// TwinCAT 3 PLC project Portal
// ProgramVersion: 3.1.4024.0
// libraries:
//   Tc2_Drive, * (Beckhoff Automation GmbH)
//   Tc2_EtherCAT, * (Beckhoff Automation GmbH)
//   Tc2_Standard, * (Beckhoff Automation GmbH)
//   Tc2_System, * (Beckhoff Automation GmbH)
//   Tc2_Utilities, * (Beckhoff Automation GmbH)
//   Tc3_Module, * (Beckhoff Automation GmbH)
// project tree:
//   DUTs/ PanelButton.TcDUT, StateMachine.TcDUT
//   POUs/ RPC_PanelProcess.TcPOU, RPC_ScopeProcess.TcPOU, RPC_SoEProcess.TcPOU, MAIN.TcPOU
//   Scope/ FB_ExportScopeData.TcPOU, FB_GenerateFileSuffixByTime.TcPOU, FB_ScopeServer.TcPOU
//   GVLs/ GlobalVar.TcGVL
//   / PlcTask.TcTTO
// real-time tasks:
//   TASK PlcTask: cycle T#250us, priority 10, ADS port 350
//   TASK MotionControl: cycle T#250us, priority 4, ADS port 352
//   TASK ModuleSpindle: cycle T#250us, priority 6, ADS port 351
//   TASK ModuleAxisGroup: cycle T#250us, priority 8, ADS port 353
//   TASK ModuleTest: cycle T#250us, priority 12, ADS port 354
//   TASK TestHMI: cycle T#10ms, priority 18, ADS port 355
//   TASK ModuleSafety: cycle T#250us, priority 14, ADS port 356
// I/O:
//   DEVICE BeckhoffBench, AmsNetId 169.254.41.58.4.1
//     ZY [AX5201-0000-0214 EtherCAT Drive (SoE, 2 Ch.)]
//     Gantry [AX5201-0000-0214 EtherCAT Drive (SoE, 2 Ch.)]
//     Panel [iA-MPA64B0 2xMII_REV00030022]
//     Drive 4 (MCDLN35BE) [MCDLN35BE]
// variable links:
//   Portal/Portal Instance <-> BeckhoffBench/Gantry
//     PlcTask Inputs/MAIN.rpc_SoEProcess.stPlcDriveRef[0]/aNetId <-> InfoData/AdsAddr/netId
//     PlcTask Inputs/MAIN.rpc_SoEProcess.stPlcDriveRef[1]/aNetId <-> InfoData/AdsAddr/netId
//     PlcTask Inputs/MAIN.rpc_SoEProcess.stPlcDriveRef[0]/nDriveNo <-> InfoData/Chn1
//     PlcTask Inputs/MAIN.rpc_SoEProcess.stPlcDriveRef[1]/nDriveNo <-> InfoData/Chn0
//     PlcTask Inputs/MAIN.rpc_SoEProcess.stPlcDriveRef[0]/nSlaveAddr <-> InfoData/AdsAddr/port
//     PlcTask Inputs/MAIN.rpc_SoEProcess.stPlcDriveRef[1]/nSlaveAddr <-> InfoData/AdsAddr/port
//   Portal/Portal Instance <-> BeckhoffBench/Panel
//     PlcTask Inputs/MAIN.rpc_PanelProcess.handwheelCurrPos <-> PANEL_Inputs/TEACH_HANDWHEEL
//     PlcTask Inputs/MAIN.rpc_PanelProcess.pInput[0] <-> PANEL_Inputs/PIO_IN1
//     PlcTask Inputs/MAIN.rpc_PanelProcess.pInput[1] <-> PANEL_Inputs/PIO_IN2
//     PlcTask Inputs/MAIN.rpc_PanelProcess.pInput[2] <-> PANEL_Inputs/PIO_IN3
//     PlcTask Inputs/MAIN.rpc_PanelProcess.pInput[3] <-> PANEL_Inputs/PIO_IN4
//     PlcTask Inputs/MAIN.rpc_PanelProcess.pInput[4] <-> PANEL_Inputs/PIO_IN5
//     PlcTask Inputs/MAIN.rpc_PanelProcess.pInput[5] <-> PANEL_Inputs/PIO_IN7
//     PlcTask Outputs/MAIN.rpc_PanelProcess.pOutput[0] <-> PANEL_Outputs/PIO_OUT1
//     PlcTask Outputs/MAIN.rpc_PanelProcess.pOutput[1] <-> PANEL_Outputs/PIO_OUT2
//     PlcTask Outputs/MAIN.rpc_PanelProcess.pOutput[2] <-> PANEL_Outputs/PIO_OUT3
//     PlcTask Outputs/MAIN.rpc_PanelProcess.pOutput[3] <-> PANEL_Outputs/PIO_OUT4
//     PlcTask Outputs/MAIN.rpc_PanelProcess.pOutput[4] <-> PANEL_Outputs/PIO_OUT5
//     PlcTask Outputs/MAIN.rpc_PanelProcess.pOutput[5] <-> PANEL_Outputs/PIO_OUT7
//   Portal/Portal Instance <-> BeckhoffBench/ZY
//     PlcTask Inputs/MAIN.rpc_SoEProcess.stPlcDriveRef[2]/aNetId <-> InfoData/AdsAddr/netId
//     PlcTask Inputs/MAIN.rpc_SoEProcess.stPlcDriveRef[3]/aNetId <-> InfoData/AdsAddr/netId
//     PlcTask Inputs/MAIN.rpc_SoEProcess.stPlcDriveRef[2]/nDriveNo <-> InfoData/Chn1
//     PlcTask Inputs/MAIN.rpc_SoEProcess.stPlcDriveRef[3]/nDriveNo <-> InfoData/Chn0
//     PlcTask Inputs/MAIN.rpc_SoEProcess.stPlcDriveRef[2]/nSlaveAddr <-> InfoData/AdsAddr/port
//     PlcTask Inputs/MAIN.rpc_SoEProcess.stPlcDriveRef[3]/nSlaveAddr <-> InfoData/AdsAddr/port
//   Portal/Portal Instance <-> MotionControl/MotionControl_Obj1 (MotionControl)
//     PlcTask Outputs/MAIN.rpc_PanelProcess.objID <-> Inputs/OidPanelProcess
//     PlcTask Outputs/MAIN.rpc_PanelProcess.panelInfoOutput <-> Inputs/PanelInformation
//     PlcTask Outputs/MAIN.rpc_ScopeProcess.objID <-> Inputs/OidScopeProcess
//   Portal/Portal Instance <-> MotionControl/MotionControl_Obj3 (ModuleAxisGroup)
//     PlcTask Outputs/MAIN.rpc_SoEProcess.objID <-> Inputs/OidSoEProcess
//   MotionControl/MotionControl_Obj1 (MotionControl) <-> MotionControl/MotionControl_Obj3 (ModuleAxisGroup)
//     Outputs/ContinuousMovingCommand <-> Inputs/ContinuousMovingCommand
//     Outputs/ManualMovingCommand <-> Inputs/ManualMovingCommand
//   MotionControl/MotionControl_Obj1 (MotionControl) <-> MotionControl/MotionControl_Obj4 (ModuleSafety)
//     Inputs/ErrorCode <-> Outputs/ErrorCode
//   MotionControl/MotionControl_Obj2 (ModuleSpindle) <-> MotionControl/MotionControl_Obj4 (ModuleSafety)
//     Outputs/SpindleInfo <-> Inputs/DiagnosticInfo/SpindleInfo
//     Outputs/StateSpindle <-> Inputs/DiagnosticInfo/StateSpindle
//   MotionControl/MotionControl_Obj3 (ModuleAxisGroup) <-> MotionControl/MotionControl_Obj4 (ModuleSafety)
//     Outputs/AxisGroupInfo <-> Inputs/DiagnosticInfo/AxisGroupInfo
//     Outputs/StateAxisGroup <-> Inputs/DiagnosticInfo/StateAxisGroup
//   (this object) <-> MotionControl/MotionControl_Obj2 (ModuleSpindle)
//     Drive 4 (MCDLN35BE)/Receive PDO mapping 1/Controlword <-> Outputs/SpindleOutput/ControlWord
//     Drive 4 (MCDLN35BE)/Receive PDO mapping 1/Modes of operation <-> Outputs/SpindleOutput/OperationMode
//     Drive 4 (MCDLN35BE)/Receive PDO mapping 1/Target position <-> Outputs/SpindleOutput/TargetPosition
//     Drive 4 (MCDLN35BE)/Transmit PDO mapping 1/Modes of operation display <-> Inputs/SpindleInput/ActualOpMode
//     Drive 4 (MCDLN35BE)/Transmit PDO mapping 1/Position actual value <-> Inputs/SpindleInput/ActualAbsPos
//     Drive 4 (MCDLN35BE)/Transmit PDO mapping 1/Statusword <-> Inputs/SpindleInput/StatusWord
//   (this object) <-> MotionControl/MotionControl_Obj3 (ModuleAxisGroup)
//     Gantry/AT 1/Class 1 diagnostic (C1D) <-> Inputs/AxisInputs[1]/ErrorCode
//     Gantry/AT 2/Class 1 diagnostic (C1D) <-> Inputs/AxisInputs[0]/ErrorCode
//     Gantry/AT 1/Drive status word <-> Inputs/AxisInputs[1]/StatusWord
//     Gantry/AT 2/Drive status word <-> Inputs/AxisInputs[0]/StatusWord
//     Gantry/AT 1/Position feedback 1 value (motor feedback) <-> Inputs/AxisInputs[1]/ActualAbsPos
//     Gantry/AT 2/Position feedback 1 value (motor feedback) <-> Inputs/AxisInputs[0]/ActualAbsPos
//     Gantry/AT 1/Torque/force feedback value <-> Inputs/AxisInputs[1]/ActualTor
//     Gantry/AT 2/Torque/force feedback value <-> Inputs/AxisInputs[0]/ActualTor
//     Gantry/AT 1/Velocity feedback 1 value <-> Inputs/AxisInputs[1]/ActualVel
//     Gantry/AT 2/Velocity feedback 1 value <-> Inputs/AxisInputs[0]/ActualVel
//     Gantry/MDT 1/Master control word <-> Outputs/AxisOutputs[1]/ControlWord
//     Gantry/MDT 2/Master control word <-> Outputs/AxisOutputs[0]/ControlWord
//     Gantry/MDT 1/Position command value <-> Outputs/AxisOutputs[1]/TargetPosition
//     Gantry/MDT 2/Position command value <-> Outputs/AxisOutputs[0]/TargetPosition
//     Gantry/MDT 1/Torque/force command value <-> Outputs/AxisOutputs[1]/TargetTorque
//     Gantry/MDT 2/Torque/force command value <-> Outputs/AxisOutputs[0]/TargetTorque
//     Gantry/MDT 1/Velocity command value <-> Outputs/AxisOutputs[1]/TargetVelocity
//     Gantry/MDT 2/Velocity command value <-> Outputs/AxisOutputs[0]/TargetVelocity
//     ZY/AT 1/Class 1 diagnostic (C1D) <-> Inputs/AxisInputs[3]/ErrorCode
//     ZY/AT 2/Class 1 diagnostic (C1D) <-> Inputs/AxisInputs[2]/ErrorCode
//     ZY/AT 1/Drive status word <-> Inputs/AxisInputs[3]/StatusWord
//     ZY/AT 2/Drive status word <-> Inputs/AxisInputs[2]/StatusWord
//     ZY/AT 1/Position feedback 1 value (motor feedback) <-> Inputs/AxisInputs[3]/ActualAbsPos
//     ZY/AT 2/Position feedback 1 value (motor feedback) <-> Inputs/AxisInputs[2]/ActualAbsPos
//     ZY/AT 1/Torque/force feedback value <-> Inputs/AxisInputs[3]/ActualTor
//     ZY/AT 2/Torque/force feedback value <-> Inputs/AxisInputs[2]/ActualTor
//     ZY/AT 1/Velocity feedback 1 value <-> Inputs/AxisInputs[3]/ActualVel
//     ZY/AT 2/Velocity feedback 1 value <-> Inputs/AxisInputs[2]/ActualVel
//     ZY/MDT 1/Additive torque/force command value <-> Outputs/AxisOutputs[3]/AdditiveTorque
//     ZY/MDT 1/Master control word <-> Outputs/AxisOutputs[3]/ControlWord
//     ZY/MDT 2/Master control word <-> Outputs/AxisOutputs[2]/ControlWord
//     ZY/MDT 1/Position command value <-> Outputs/AxisOutputs[3]/TargetPosition
//     ZY/MDT 2/Position command value <-> Outputs/AxisOutputs[2]/TargetPosition
//     ZY/MDT 1/Torque/force command value <-> Outputs/AxisOutputs[3]/TargetTorque
//     ZY/MDT 2/Torque/force command value <-> Outputs/AxisOutputs[2]/TargetTorque
//     ZY/MDT 1/Velocity command value <-> Outputs/AxisOutputs[3]/TargetVelocity
//     ZY/MDT 2/Velocity command value <-> Outputs/AxisOutputs[2]/TargetVelocity
//   (this object) <-> MotionControl/MotionControl_Obj4 (ModuleSafety)
//     Gantry/AT 1/Digital inputs, state <-> Inputs/DiagnosticInfo/AxisGroupDigitalInput[1]
//     Gantry/AT 2/Digital inputs, state <-> Inputs/DiagnosticInfo/AxisGroupDigitalInput[0]
//     ZY/AT 1/Digital inputs, state <-> Inputs/DiagnosticInfo/AxisGroupDigitalInput[3]
//     ZY/AT 2/Digital inputs, state <-> Inputs/DiagnosticInfo/AxisGroupDigitalInput[2]
//   TestHMI Instance <-> ModuleTest/ModuleTest_Obj1 (ModuleTest)
//     TestHMI Outputs/MAIN.MockPanel <-> Inputs/MockPanel
//     TestHMI Outputs/MAIN.Recovery <-> Inputs/RecoveryButton
//   TestHMI Instance <-> MotionControl/MotionControl_Obj1 (MotionControl)
//     TestHMI Inputs/MAIN.TestMainState <-> Outputs/MainState
//   TestHMI Instance <-> MotionControl/MotionControl_Obj2 (ModuleSpindle)
//     TestHMI Inputs/MAIN.TestSpindleState <-> Outputs/StateSpindle
//   TestHMI Instance <-> MotionControl/MotionControl_Obj3 (ModuleAxisGroup)
//     TestHMI Inputs/MAIN.TestAxisGroupState <-> Outputs/StateAxisGroup
//   TestHMI Instance <-> MotionControl/MotionControl_Obj4 (ModuleSafety)
//     TestHMI Inputs/MAIN.TestSafetyStatus <-> Outputs/SafetyStatus

CONFIGURATION Portal
    RESOURCE PLC ON TwinCAT3
        TASK PlcTask(INTERVAL := T#250us, PRIORITY := 10);
        PROGRAM MAIN WITH PlcTask : MAIN;
    END_RESOURCE
END_CONFIGURATION

// ---- DUTs/PanelButton.TcDUT
TYPE PanelButton :
STRUCT
	alias   : STRING;
	pressed : BOOL;
	row   	: INT;
	column 	: INT;
END_STRUCT
END_TYPE

// ---- DUTs/StateMachine.TcDUT
TYPE StateMachine :
STRUCT
	AxisGroupState : SystemState;
	SpindleState : SystemState;
END_STRUCT
END_TYPE

// ---- GVLs/GlobalVar.TcGVL
VAR_GLOBAL CONSTANT
	// Scope server related
	RECORD_CONFIG_PATH 		: STRING := 'C:/RecordData/ScopeServer/RecordData.tcscopex';
	RECORD_CONFIG_XML_PATH 	: STRING := 'C:/RecordData/Settings/ScopeExporterSettings.xml';
	SAVE_SVDX_PREFIX 		: STRING := 'C:/RecordData/SVDX/'; 
	SAVE_CSV_PREFIX			: STRING := 'C:/RecordData/CSV/'; 
	
	// Motion Control
	MC_AXIS_NUM    : INT := 5;
	MAX_DRIVER_NUM : INT := 10;
	ACTIVE_DRIVER_NUM : INT := 4;
	
	// Panel Information
	PANEL_CHANNEL_NUM   :INT := 6;
	CHANNEL_BUTTON_NUM  :INT := 8;
	HANDWHEEL_FULL_SCALE :INT := 256;
	RESET_DURATION :INT := 10;
END_VAR

// Define buttons of panel to improve code readability
VAR_GLOBAL
	ServoOn 			: PanelButton;
	X_Axis  			: PanelButton;
	Y_Axis  			: PanelButton;
	Z_Axis  			: PanelButton;
	A_Axis  			: PanelButton;
	B_Axis  			: PanelButton;
	C_Axis  			: PanelButton;
	Spindle_CW			: PanelButton;
	Spindle_CCW			: PanelButton;
	Spindle_Stop		: PanelButton;
	Spindle_Direct      : PanelButton;
	Tenth_Ratio   		: PanelButton;
	Hundredth_Ratio   	: PanelButton;
	Thousandth_Ratio   	: PanelButton;
	Reset_Button        : PanelButton;
	Execute_Button      : PanelButton;
	Cyclical_Run        : PanelButton;
END_VAR

// ---- POUs/MAIN.TcPOU
PROGRAM MAIN
VAR
	bInit 	  : BOOL := FALSE; // flag for initialization
	bTaskDone : BOOL := FALSE;
END_VAR
	
// Scope Server
VAR
	fb_GenerateFileSuffixByTime : FB_GenerateFileSuffixByTime; 	// Generate file suffix by system time
	fb_ScopeServer 		  		: FB_ScopeServer; 	  			// Record .svdx file
	bScopeRun 			  		: BOOL := FALSE; 		  		// Flag of starting or stoping scope server
	fb_ExportScopeData 	  		: FB_ExportScopeData;   		// Export recorded data after finishing 
	bExportData    		  		: BOOL := FALSE; 		  		// Flag of exporting data to file
END_VAR

// RPC module
VAR
	rpc_SoEProcess : RPC_SoEProcess('MAIN.rpc_SoEProcess');
	rpc_PanelProcess : RPC_PanelProcess('MAIN.rpc_PanelProcess');
	rpc_ScopeProcess : RPC_ScopeProcess('MAIN.rpc_ScopeProcess');
END_VAR

rpc_ScopeProcess();

END_PROGRAM

// ---- Scope/FB_GenerateFileSuffixByTime.TcPOU
FUNCTION_BLOCK FB_GenerateFileSuffixByTime
VAR
	fb_LocalSystemTime 	: FB_LocalSystemTime; // function provided by beckhoff to get system time
	fb_FormatString		: FB_FormatString;    // function provided by beckhoff to convert arguments in a string and format them
END_VAR

VAR
	year		: DINT;
	month		: DINT;
	day			: DINT;
	hour		: DINT;
	minute      : DINT;
	lastHour	: DINT;
	formatDate	: T_MaxString;
	
	SAVE_SVDX_SUFFIX : STRING;
	SAVE_CSV_SUFFIX  : STRING;
END_VAR

// Enable time synchronization
fb_LocalSystemTime.bEnable := TRUE;	

// Get current local time
fb_LocalSystemTime();
year 	:= DWORD_TO_DINT(fb_LocalSystemTime.systemTime.wYear);
month 	:= DWORD_TO_DINT(fb_LocalSystemTime.systemTime.wMonth);
day 	:= DWORD_TO_DINT(fb_LocalSystemTime.systemTime.wDay);
hour 	:= DWORD_TO_DINT(fb_LocalSystemTime.systemTime.wHour);
minute 	:= DWORD_TO_DINT(fb_LocalSystemTime.systemTime.wMinute);

fb_FormatString(sFormat := '%.4d%.2d%.2d%.2d%.2d',
				arg1 := F_DINT(year),
				arg2 := F_DINT(month),
				arg3 :=	F_DINT(day),
				arg4 :=	F_DINT(hour),
				arg5 :=	F_DINT(minute),
				sOut => formatDate);

// Generate suffix of file to be saved				
SAVE_SVDX_SUFFIX := CONCAT(formatDate, '.svdx');
SAVE_CSV_SUFFIX := CONCAT(formatDate, '.CSV');

END_FUNCTION_BLOCK

// ---- Scope/FB_ScopeServer.TcPOU
FUNCTION_BLOCK FB_ScopeServer
VAR_INPUT
	//sNetId					: STRING	:='';	
    bExternalTriggerEvent	: BOOL 	:= FALSE; //Rising edge start recording, falling edge stop and save
	sConfigFile				: STRING; //.tcscopex
	sSaveFile				: STRING; //.svdx
END_VAR
//VAR_OUTPUT
VAR
    bBusy					: BOOL 		:= FALSE;
    bError					: BOOL 		:= FALSE;
    nErrorId				: UDINT 	:= 0;	
END_VAR
VAR

    bDone					: BOOL 		:= FALSE;	

    fbScopeServerControl	: FB_ScopeServerControl;
    eReqState				: E_ScopeServerState := SCOPE_SERVER_IDLE;
	
    eState					: (IDLE,RECORDING,SAVING,DISCONNECTING,ERROR,RESETING);
END_VAR

CASE eState OF
	IDLE:
		bBusy	:=FALSE;
		IF bExternalTriggerEvent THEN
			bBusy			:= TRUE;
	    	eReqState 		:= SCOPE_SERVER_START;
	    	eState 			:= RECORDING;	
		END_IF
	
	RECORDING:	
		IF fbScopeServerControl.bDone THEN
	    	IF NOT bExternalTriggerEvent THEN
	    	    eReqState 		:= SCOPE_SERVER_SAVE;
	    	    eState 			:= SAVING;
	    	END_IF
		ELSIF fbScopeServerControl.bError THEN
			eState	:=ERROR;		
		END_IF
		
	SAVING:
	    IF fbScopeServerControl.bDone THEN
	        eReqState 		:= SCOPE_SERVER_DISCONNECT;
			eState			:= DISCONNECTING;
		ELSIF fbScopeServerControl.bError THEN
			eState	:=ERROR;		
		END_IF
		
	DISCONNECTING:
		IF fbScopeServerControl.bDone THEN
	       eState := IDLE;
		ELSIF fbScopeServerControl.bError THEN
			eState	:=ERROR;				   
	    END_IF		
		
	ERROR:
		bBusy			:= FALSE;
		IF NOT bExternalTriggerEvent THEN
			bBusy			:= TRUE;
			eReqState 		:= SCOPE_SERVER_RESET;
			eState			:= DISCONNECTING;
		END_IF
		
	RESETING:
		IF fbScopeServerControl.bDone OR fbScopeServerControl.bError THEN
	       	eReqState 		:= SCOPE_SERVER_IDLE;
			eState			:= IDLE; 
	    END_IF		
		
END_CASE


fbScopeServerControl( sNetId		:= '',
                      eReqState		:= eReqState,
                      sConfigFile	:= sConfigFile,
                      sSaveFile		:= sSaveFile,
                      tTimeout		:= T#10S,
                      bBusy			=>,
                      bDone			=>bDone,
                      bError		=>bError,
                      nErrorId		=>nErrorId);

END_FUNCTION_BLOCK

// ---- Scope/FB_ExportScopeData.TcPOU
FUNCTION_BLOCK FB_ExportScopeData
VAR_INPUT
	sNetId			:STRING	:='';	
	bExport			:BOOL;
	svd 			:T_MaxString; //.svdx
	target			:T_MaxString; //.csv
	config			:T_MaxString; //.xml Configuration file created by export wizzard
	Channellist		:T_MaxString; //Channel List (Names of the channels(s) separated with semicolon
	start			:T_MaxString; //Starttime (As TwinCAT time stamp)
	end				:T_MaxString; //Endtime (As TwimCAT time stamp	
END_VAR
//VAR_OUTPUT
VAR
	bBusy			:BOOL;
	bError			:BOOL;
	iErrorID		:UDINT;
END_VAR
VAR
	rtExport		:R_TRIG; // Detect rising edge
	fbStartExport	:NT_StartProcess;
	
	eState			:(IDLE,EXPORTING,ERROR);
	
    fbFormat   		: FB_FormatString2;
    sFormat    		: T_MaxString ;
	sCommand		: T_MaxString ;
END_VAR

rtExport(CLK:=bExport);
CASE eState OF 
	IDLE:
		bBusy		:=FALSE;
		IF rtExport.Q THEN
			bBusy		:=TRUE;
			sFormat:='"svd=%s" "target=%s"';
			
			IF config<>'' THEN
				sFormat:= CONCAT(sFormat,' "config=%s"');
			ELSE
				sFormat:= CONCAT(sFormat,'%s');
			END_IF

			IF Channellist<>'' THEN
				sFormat:= CONCAT(sFormat,' "Channellist=%s"');
			ELSE
				sFormat:= CONCAT(sFormat,'%s');
			END_IF
			
			IF start<>'' THEN
				sFormat:= CONCAT(sFormat,' "start=%s"');
			ELSE
				sFormat:= CONCAT(sFormat,'%s');
			END_IF			

			IF end<>'' THEN
				sFormat:= CONCAT(sFormat,' "end=%s"');
			ELSE
				sFormat:= CONCAT(sFormat,'%s');
			END_IF					
			
			sFormat	:= CONCAT(sFormat,' silent');
			
			fbFormat(
				pFormatString:=ADR(sFormat) , 
				arg1		:=F_STRING(svd) , 
				arg2		:=F_STRING(target) ,
				arg3		:=F_STRING(config), 
				arg4		:=F_STRING(Channellist), 
				arg5		:=F_STRING(start), 
				arg6		:=F_STRING(end), 				
				arg7		:=, 				
				pDstString	:=ADR(sCommand) , 
				nDstSize	:=SIZEOF(sCommand) );
				
			IF NOT fbFormat.bError THEN
				eState				:=EXPORTING;
				fbStartExport.START	:=TRUE;
			ELSE
				bError		:=fbFormat.bError;
				iErrorID	:=fbFormat.nErrId;
				eState		:=ERROR;
			END_IF
			
		END_IF
	
	EXPORTING:
		IF NOT fbStartExport.BUSY THEN
			fbStartExport.START	:=FALSE;
			IF NOT fbStartExport.ERR THEN
				eState		:=IDLE;
			ELSE
				bError		:=fbStartExport.ERR;
				iErrorID	:=fbStartExport.ERRID;
				eState		:=ERROR;				
			END_IF
		END_IF
	
	ERROR:
		eState		:=IDLE;
		
END_CASE


fbStartExport(
    NETID		:= sNetId, 
    PATHSTR		:= 'C:\TwinCAT\Functions\TE130X-Scope-View\TC3ScopeExportTool.exe', 
    DIRNAME		:= 'C:\TwinCAT\Functions\TE130X-Scope-View', 
    COMNDLINE	:= sCommand, 
    START		:= , 
    TMOUT		:= T#30S);

END_FUNCTION_BLOCK

// ---- POUs/RPC_SoEProcess.TcPOU
{attribute 'c++_compatible'}
FUNCTION_BLOCK RPC_SoEProcess EXTENDS TcBaseModuleRegistered IMPLEMENTS ISoEProcess

VAR
	fbSoEReset : ARRAY [0..GlobalVar.MAX_DRIVER_NUM-1] OF FB_SoEReset_ByDriveRef; //SoE Reset
	fbSoEWrite : ARRAY [0..GlobalVar.MAX_DRIVER_NUM-1] OF FB_SoEWrite_ByDriveRef; //SoE Write
	fbSoERead : ARRAY [0..GlobalVar.MAX_DRIVER_NUM-1] OF FB_SoERead_ByDriveRef; //SoE Read
	stPlcDriveRef AT %I* : ARRAY [0..GlobalVar.MAX_DRIVER_NUM-1] OF ST_PlcDriveRef;
	stDriveRef : ARRAY [0..GlobalVar.MAX_DRIVER_NUM-1] OF ST_DriveRef;
	bBusyFlag : ARRAY  [0..GlobalVar.MAX_DRIVER_NUM-1] OF BOOL;
END_VAR

METHOD FB_reinit : BOOL
VAR_INPUT
END_VAR
SUPER^.FB_reinit();
END_METHOD

{attribute 'object_name' := 'mInitialize'}
{attribute 'c++_compatible'}
{attribute 'minimal_input_size' := '4'}
{attribute 'pack_mode' := '4'}
{attribute 'show'}
{attribute 'checksuperglobal'}

METHOD mInitialize : HRESULT

VAR
	loopDriver 	: INT := 0;
	tempRet     : HRESULT;
END_VAR
mInitialize := S_FALSE;

FOR loopDriver := 0 TO GlobalVar.ACTIVE_DRIVER_NUM - 1 DO
		stDriveRef[loopDriver].sNetId  := F_CreateAmsNetId(stPlcDriveRef[loopDriver].aNetId); // convert the byte array into a string
		stDriveRef[loopDriver].nSlaveAddr := stPlcDriveRef[loopDriver].nSlaveAddr;
		stDriveRef[loopDriver].nDriveNo := stPlcDriveRef[loopDriver].nDriveNo;
		stDriveRef[loopDriver].nDriveType := stPlcDriveRef[loopDriver].nDriveType;
END_FOR

FOR loopDriver := 0 TO GlobalVar.ACTIVE_DRIVER_NUM - 1 DO
	tempRet := S_FALSE;
	IF (stDriveRef[loopDriver].sNetId <> '') AND (stDriveRef[loopDriver].nSlaveAddr <> 0) THEN
		tempRet := S_OK;
	END_IF
	mInitialize := tempRet AND S_OK;
END_FOR
END_METHOD

{attribute 'object_name' := 'mReset'}
{attribute 'c++_compatible'}
{attribute 'minimal_input_size' := '4'}
{attribute 'pack_mode' := '4'}
{attribute 'show'}
{attribute 'checksuperglobal'}

METHOD mReset : HRESULT
VAR_INPUT
	bExecute	: BOOL;
END_VAR
VAR
	loopDriver 	: INT := 0;
	tempRet     : HRESULT;
END_VAR
mReset := S_FALSE;

IF bExecute THEN
	FOR loopDriver := 0 TO GlobalVar.ACTIVE_DRIVER_NUM - 1 DO 
		fbSoEReset[loopDriver](stDriveRef := stDriveRef[loopDriver], 
									bExecute := TRUE, tTimeout := TIME#10S,
									bBusy=>bBusyFlag[loopDriver], bError=>, iAdsErrId=>, iSercosErrId=>);
		tempRet := S_FALSE;
		IF NOT bBusyFlag[loopDriver] THEN // This output is set when the function block is activated, and remains set until a feedback is received.
			fbSoEReset[loopDriver](stDriveRef := stDriveRef[loopDriver], bExecute := FALSE);				
			tempRet := S_OK;
		END_IF
		mReset := tempRet AND S_OK;
	END_FOR
END_IF
END_METHOD

{attribute 'TcTypeSystem'}
{attribute 'no-analysis'}
{attribute 'c++_compatible'}
{attribute 'minimal_input_size' := '4'}
{attribute 'pack_mode' := '4'}

METHOD mSoEWritePositionLoopKv : HRESULT
VAR_INPUT
	axis	: INT;
	value	: REAL;
END_VAR
END_METHOD

{attribute 'TcTypeSystem'}
{attribute 'no-analysis'}
{attribute 'c++_compatible'}
{attribute 'minimal_input_size' := '4'}
{attribute 'pack_mode' := '4'}

METHOD mSoEWriteVelocityLoopKp : HRESULT
VAR_INPUT
	axis	: INT;
	value	: REAL;
END_VAR
fbSoEWrite[axis](stDriveRef := stDriveRef[axis],
				nIdn := S_0_IDN + 100, // S-0-0100 Velocity loop proportional gain
				nElement := 16#40, // Value element
				pSrcBuf := ADR(value),
				cbBufLen := SIZEOF(value),
				bExecute := TRUE,
				tTimeOut := DEFAULT_ADS_TIMEOUT);
				
IF NOT fbSoEWrite[axis].bBusy THEN
	IF NOT fbSoEWrite[axis].bError THEN 
        (* write successful *)
       fbSoEWrite[axis](bExecute := FALSE);
    END_IF 
END_IF
END_METHOD

{attribute 'object_name' := 'TcQueryInterface'}
{attribute 'c++_compatible'}
{attribute 'minimal_input_size' := '4'}
{attribute 'pack_mode' := '4'}
{attribute 'show'}
{attribute 'checksuperglobal'}

METHOD TcQueryInterface : HRESULT
VAR_INPUT
	iid	: REFERENCE TO IID;
	pipItf	: POINTER TO PVOID;
END_VAR

VAR
	ipSoE : ISoEProcess;
	ipUnk : ITcUnknown;
END_VAR
IF GuidsEqual(ADR(iid), ADR(TC_GLOBAL_IID_LIST.IID_ISoEProcess)) THEN
	ipSoE := THIS^; // cast to interface pointer
	pipItf^ := ITCUNKNOWN_TO_PVOID(ipSoE);
	TcAddRef();
	TcQueryInterface := S_OK;
ELSIF GuidsEqual(ADR(iid), ADR(TC_GLOBAL_IID_LIST.IID_ITcUnknown)) THEN
	ipUnk := THIS^; // cast to interface pointer
	pipItf^ := ITCUNKNOWN_TO_PVOID(ipUnk);
	TcAddRef(); 
	TcQueryInterface := S_OK;
ELSE
	TcQueryInterface := SUPER^.TcQueryInterface(iid, pipItf);
END_IF
END_METHOD

END_FUNCTION_BLOCK

// ---- POUs/RPC_PanelProcess.TcPOU
{attribute 'c++_compatible'}
FUNCTION_BLOCK RPC_PanelProcess EXTENDS TcBaseModuleRegistered IMPLEMENTS IPanelProcess
VAR
	pInput AT%I* : ARRAY[0..GlobalVar.PANEL_CHANNEL_NUM-1] OF USINT; // Connect to panel input channel 1 2 3 4 5 7 
	pOutput AT%Q* : ARRAY[0..GlobalVar.PANEL_CHANNEL_NUM-1] OF USINT; // Connect to panel output channel 1 2 3 4 5 7
	lastInput : ARRAY[0..GlobalVar.PANEL_CHANNEL_NUM-1] OF USINT; // Record input channel value of last cycle
	valChanged : ARRAY[0..GlobalVar.PANEL_CHANNEL_NUM-1] OF BOOL; // used in button mutex check since some mutex pairs appear in different channels 
	
	// Decompose value of input channel into status of single button, one channel represents eight buttons
	buttonStatus : ARRAY[0..GlobalVar.PANEL_CHANNEL_NUM-1,0..GlobalVar.CHANNEL_BUTTON_NUM-1] OF BOOL := [FALSE]; 
	effectiveButtonStatus : ARRAY[0..GlobalVar.PANEL_CHANNEL_NUM-1,0..GlobalVar.CHANNEL_BUTTON_NUM-1] OF BOOL := [FALSE];
	
	mutexPairs: ARRAY[0..30, 0..1] OF PanelButton; // 30 represents the maximum number of possible pairs
	mutexPairNum : INT := 0;
END_VAR

// HandWheel Functions
VAR
	handwheelCurrPos 	AT%I* :  USINT;
	handwheelLastPos 	: USINT;
	handwheelTotalPos : ARRAY[0..GlobalVar.MC_AXIS_NUM - 1] OF LREAL := [0.0]; // X Y Z A C
	
	panelInfoOutput AT%Q* : PanelInfo; // Necessary information sent to Cpp module
END_VAR

// Special button handle
VAR
	iResetCount :INT := 0;
	bSpindleStopSet       : BOOL := FALSE;
END_VAR

METHOD FB_reinit : BOOL
VAR_INPUT
END_VAR
SUPER^.FB_reinit();
END_METHOD

METHOD mAssignSpecifcButtonCoordinate : BOOL
VAR_INPUT
END_VAR
ServoOn.row := 0;
ServoOn.column := 0;

X_Axis.row := 0;  
X_Axis.column := 6;  

Y_Axis.row := 0;  
Y_Axis.column := 7;

Z_Axis.row := 1;  
Z_Axis.column := 0;  

A_Axis.row := 1;  
A_Axis.column := 7;  

B_Axis.row := 2;  
B_Axis.column := 0;  

C_Axis.row := 2;  
C_Axis.column := 1;  

Spindle_CW.row := 2;
Spindle_CW.column := 2;

Spindle_CCW.row := 2;
Spindle_CCW.column := 4;

Spindle_Stop.row := 2;
Spindle_Stop.column	:= 3;

Spindle_Direct.row := 4;
Spindle_Direct.column := 0;
	
Tenth_Ratio.row := 4;  
Tenth_Ratio.column := 1;  
 
Hundredth_Ratio.row := 4;
Hundredth_Ratio.column := 2;

Thousandth_Ratio.row := 4;
Thousandth_Ratio.column := 3;

Reset_Button.row := 5;
Reset_Button.column := 0;

Execute_Button.row := 5;
Execute_Button.column := 1;

Cyclical_Run.row := 5;
Cyclical_Run.column := 2;

mGenerateMutexPair(X_Axis, Y_Axis);
mGenerateMutexPair(X_Axis, Z_Axis);
mGenerateMutexPair(X_Axis, A_Axis);
mGenerateMutexPair(X_Axis, B_Axis);
mGenerateMutexPair(X_Axis, C_Axis);
                                 
mGenerateMutexPair(Y_Axis, Z_Axis);
mGenerateMutexPair(Y_Axis, A_Axis);
mGenerateMutexPair(Y_Axis, B_Axis);
mGenerateMutexPair(Y_Axis, C_Axis);
                                 
mGenerateMutexPair(Z_Axis, A_Axis);
mGenerateMutexPair(Z_Axis, B_Axis);
mGenerateMutexPair(Z_Axis, C_Axis);
                                 
mGenerateMutexPair(A_Axis, B_Axis);
mGenerateMutexPair(A_Axis, C_Axis);
mGenerateMutexPair(B_Axis, C_Axis);

mGenerateMutexPair(Tenth_Ratio, Hundredth_Ratio);
mGenerateMutexPair(Tenth_Ratio, Thousandth_Ratio);
mGenerateMutexPair(Hundredth_Ratio, Thousandth_Ratio);

mGenerateMutexPair(Reset_Button, Execute_Button);
mGenerateMutexPair(Reset_Button, Cyclical_Run);
END_METHOD

{attribute 'TcTypeSystem'}
{attribute 'no-analysis'}
{attribute 'c++_compatible'}
{attribute 'minimal_input_size' := '4'}
{attribute 'pack_mode' := '4'}
METHOD mDeselectAxis : HRESULT
mDeselectAxis := S_FALSE;

mPopButton(X_Axis);
mPopButton(Y_Axis);
mPopButton(Z_Axis);
mPopButton(A_Axis);
mPopButton(C_Axis);

mPopButton(Tenth_Ratio);
mPopButton(Hundredth_Ratio);
mPopButton(Thousandth_Ratio);

handwheelLastPos := handwheelCurrPos;

MEMSET(ADR(handwheelTotalPos),0, SIZEOF(handwheelTotalPos));

MEMSET(ADR(panelInfoOutput.Handwheel_EnabledAxisNum),0,SIZEOF(panelInfoOutput.Handwheel_EnabledAxisNum));
	
MEMSET(ADR(panelInfoOutput.Handwheel_dPos),0,SIZEOF(PanelInfo.Handwheel_dPos));

mDeselectAxis := S_OK;
END_METHOD

{attribute 'TcTypeSystem'}
{attribute 'no-analysis'}
{attribute 'c++_compatible'}
{attribute 'minimal_input_size' := '4'}
{attribute 'pack_mode' := '4'}

METHOD mFaultReset : HRESULT
// When system state falls into Fault, turn off all buttons for safety
MEMSET(ADR(effectiveButtonStatus), 0, SIZEOF(effectiveButtonStatus));
MEMSET(ADR(valChanged) ,0, SIZEOF(valChanged));
MEMSET(ADR(lastInput), 0, SIZEOF(lastInput));
MEMSET(ADR(pInput), 0, SIZEOF(pInput));
MEMSET(ADR(pOutput), 0, SIZEOF(pOutput));
bSpindleStopSet := FALSE;

mFaultReset := S_OK;
END_METHOD

METHOD mGenerateMutexPair : BOOL
VAR_INPUT
	button1 : PanelButton;
	button2 : PanelButton;
END_VAR
mutexPairs[mutexPairNum,0] := button1;
mutexPairs[mutexPairNum,1] := button2;

mutexPairNum := mutexPairNum + 1;
END_METHOD

METHOD mGetButtonStatus : BOOL
VAR_INPUT
END_VAR
mGetServoButtonStatus();

mGetExecuteButtonStatus();

mGetHandWheelRatio();

mGetHandwheelEnabledAxis();

mGetSpindleButtonStatus();

mGetResetButtonStatus();
END_METHOD

METHOD mGetExecuteButtonStatus : BOOL
VAR_INPUT
END_VAR
Execute_Button.pressed := effectiveButtonStatus[Execute_Button.row, Execute_Button.column];

IF Execute_Button.pressed THEN
	panelInfoOutput.Execute := TRUE;

ELSE	
	panelInfoOutput.Execute := FALSE;
END_IF
END_METHOD

METHOD mGetHandwheelEnabledAxis : BOOL
VAR_INPUT
END_VAR
X_Axis.pressed := effectiveButtonStatus[X_Axis.row, X_Axis.column];
Y_Axis.pressed := effectiveButtonStatus[Y_Axis.row, Y_Axis.column];
Z_Axis.pressed := effectiveButtonStatus[Z_Axis.row, Z_Axis.column];
A_Axis.pressed := effectiveButtonStatus[A_Axis.row, A_Axis.column];
C_Axis.pressed := effectiveButtonStatus[C_Axis.row, C_Axis.column];

// Assume no axis selected
panelInfoOutput.Handwheel_EnabledAxisNum := 0;

IF X_Axis.pressed THEN // X axis selected; 
	panelInfoOutput.Handwheel_EnabledAxisNum := AxisOrder.Axis_X;
ELSIF Y_Axis.pressed THEN // Y axis selected
	panelInfoOutput.Handwheel_EnabledAxisNum := AxisOrder.Axis_Y;	
ELSIF Z_Axis.pressed THEN // Z axis selected
	panelInfoOutput.Handwheel_EnabledAxisNum := AxisOrder.Axis_Z;
ELSIF A_Axis.pressed THEN // A axis selected
	panelInfoOutput.Handwheel_EnabledAxisNum := AxisOrder.Axis_A;	
ELSIF C_Axis.pressed THEN // C axis selected
	panelInfoOutput.Handwheel_EnabledAxisNum := AxisOrder.Axis_C;
END_IF

IF panelInfoOutput.Handwheel_EnabledAxisNum <> 0 THEN
	mHandwheelProcess(panelInfoOutput.Handwheel_EnabledAxisNum - 1);
END_IF

handwheelLastPos := handwheelCurrPos;
END_METHOD

METHOD mGetHandwheelRatio : BOOL
VAR_INPUT
END_VAR
Tenth_Ratio.pressed := effectiveButtonStatus[Tenth_Ratio.row, Tenth_Ratio.column];
Hundredth_Ratio.pressed := effectiveButtonStatus[Hundredth_Ratio.row, Hundredth_Ratio.column];
Thousandth_Ratio.pressed := effectiveButtonStatus[Thousandth_Ratio.row, Thousandth_Ratio.column];

IF Tenth_ratio.pressed THEN
	panelInfoOutput.Handwheel_Ratio := 0.1;
ELSIF Hundredth_ratio.pressed THEN
	panelInfoOutput.Handwheel_Ratio := 0.01;
ELSIF Thousandth_ratio.pressed THEN
	panelInfoOutput.Handwheel_Ratio := 0.001;
ELSE	
	panelInfoOutput.Handwheel_Ratio := 0.0;
END_IF
END_METHOD

METHOD mGetResetButtonStatus : BOOL
VAR_INPUT
END_VAR
Reset_Button.pressed := effectiveButtonStatus[Reset_Button.row, Reset_Button.column];

IF Reset_Button.pressed THEN
	panelInfoOutput.Reset := TRUE;

ELSE	
	panelInfoOutput.Reset := FALSE;
END_IF
END_METHOD

METHOD mGetServoButtonStatus : BOOL
VAR_INPUT
END_VAR
ServoOn.pressed := effectiveButtonStatus[ServoOn.row, ServoOn.column];

IF ServoOn.pressed THEN
	panelInfoOutput.ServoOn := TRUE;

ELSE	
	panelInfoOutput.ServoOn := FALSE;
END_IF
END_METHOD

METHOD mGetSpindleButtonStatus : BOOL
VAR_INPUT
END_VAR
Spindle_CW.pressed := effectiveButtonStatus[Spindle_CW.row, Spindle_CW.column];
Spindle_CCW.pressed := effectiveButtonStatus[Spindle_CCW.row, Spindle_CCW.column];
Spindle_Stop.pressed := effectiveButtonStatus[Spindle_Stop.row, Spindle_Stop.column];

IF Spindle_CW.pressed THEN
	panelInfoOutput.Spindle_Cmd := 1;
ELSIF Spindle_CCW.pressed THEN 
	panelInfoOutput.Spindle_Cmd := -1;	
ELSIF Spindle_Stop.pressed THEN
	panelInfoOutput.Spindle_Cmd := 0;
ELSE
	panelInfoOutput.Spindle_Cmd := 0;
END_IF
END_METHOD

METHOD mHandwheelProcess : BOOL
VAR_INPUT
	index   : INT;
END_VAR

VAR
	dPos    : INT;
END_VAR
dPos := handwheelCurrPos - handwheelLastPos;

IF dPos > 100 THEN
	dPos := GlobalVar.HANDWHEEL_FULL_SCALE - dPos;
ELSIF dPos < -100 THEN
	dPos := GlobalVar.HANDWHEEL_FULL_SCALE + dPos;
END_IF

handwheelTotalPos[index] := handwheelTotalPos[index] + panelInfoOutput.Handwheel_Ratio * dPos;

panelInfoOutput.Handwheel_dPos[index] := handwheelTotalPos[index];
END_METHOD

{attribute 'TcTypeSystem'}
{attribute 'no-analysis'}
{attribute 'c++_compatible'}
{attribute 'minimal_input_size' := '4'}
{attribute 'pack_mode' := '4'}

METHOD mHandwheelReset : HRESULT
mHandwheelReset := S_FALSE;

handwheelLastPos := handwheelCurrPos;

MEMSET(ADR(handwheelTotalPos),0, SIZEOF(handwheelTotalPos));
	
MEMSET(ADR(panelInfoOutput.Handwheel_dPos),0,SIZEOF(PanelInfo.Handwheel_dPos));

mHandwheelReset := S_OK;
END_METHOD

{attribute 'TcTypeSystem'}
{attribute 'no-analysis'}
{attribute 'c++_compatible'}
{attribute 'minimal_input_size' := '4'}
{attribute 'pack_mode' := '4'}

METHOD mInitialize : HRESULT
mAssignSpecifcButtonCoordinate();

handwheelLastPos := handwheelCurrPos;

mInitialize := S_OK;
END_METHOD

{attribute 'TcTypeSystem'}
{attribute 'no-analysis'}
{attribute 'c++_compatible'}
{attribute 'minimal_input_size' := '4'}
{attribute 'pack_mode' := '4'}

METHOD mInput : HRESULT

VAR
	iLoop : INT := 0;
	jLoop : INT := 0;
END_VAR
FOR iLoop := 0 TO GlobalVar.PANEL_CHANNEL_NUM - 1 DO
	FOR jLoop := 0 TO GlobalVar.CHANNEL_BUTTON_NUM - 1 DO
		buttonStatus[iLoop, jLoop] := mParsePanelInput(pInput[iLoop], jLoop);
	END_FOR
END_FOR
END_METHOD

METHOD mMutexCheck : BOOL
VAR_IN_OUT
	currentInput 	: ARRAY[0..GlobalVar.PANEL_CHANNEL_NUM - 1,0..GlobalVar.CHANNEL_BUTTON_NUM - 1] OF BOOL;
	lastInput 		: ARRAY[0..GlobalVar.PANEL_CHANNEL_NUM - 1,0..GlobalVar.CHANNEL_BUTTON_NUM - 1] OF BOOL;
	bChanged		: ARRAY[0..GlobalVar.PANEL_CHANNEL_NUM - 1] OF BOOL;
END_VAR
VAR
	iLoop : INT;
END_VAR
FOR iLoop := 0 TO mutexPairNum - 1 DO
	mMutexCheckSub(currentInput, lastInput, bChanged, mutexPairs[iLoop,0], mutexPairs[iLoop,1]);
END_FOR
END_METHOD

METHOD mMutexCheckSub : BOOL
VAR_IN_OUT
	current : ARRAY[0..GlobalVar.PANEL_CHANNEL_NUM - 1,0..GlobalVar.CHANNEL_BUTTON_NUM - 1] OF BOOL;
	last	: ARRAY[0..GlobalVar.PANEL_CHANNEL_NUM - 1,0..GlobalVar.CHANNEL_BUTTON_NUM - 1] OF BOOL;
	bChanged: ARRAY[0..GlobalVar.PANEL_CHANNEL_NUM - 1] OF BOOL;
END_VAR

VAR_INPUT
	button1 : PanelButton;
	button2 : PanelButton;
END_VAR
IF current[button1.row,button1.column] AND last[button2.row,button2.column] THEN
	current[button2.row,button2.column] := TRUE;
	bChanged[button2.row] := TRUE;
END_IF

IF current[button2.row,button2.column] AND last[button1.row,button1.column] THEN
	current[button1.row,button1.column] := TRUE;
	bChanged[button1.row] := TRUE;
END_IF
END_METHOD

{attribute 'TcTypeSystem'}
{attribute 'no-analysis'}
{attribute 'c++_compatible'}
{attribute 'minimal_input_size' := '4'}
{attribute 'pack_mode' := '4'}

METHOD mOutput : HRESULT

VAR
	iLoop : INT := 0;
	jLoop : INT := 0;
	temp  :INT := 0;
END_VAR
mSpecialButtonHandle();

mMutexCheck(buttonStatus, effectiveButtonStatus, valChanged);

FOR iLoop := 0 TO GlobalVar.PANEL_CHANNEL_NUM - 1 DO
	FOR jLoop := 0 TO GlobalVar.CHANNEL_BUTTON_NUM - 1 DO
		
		IF (iLoop = Spindle_Stop.row AND jLoop = Spindle_Stop.column) OR
		   (iLoop = Spindle_CCW.row AND jLoop = Spindle_CCW.column) OR
 		   (iLoop = Spindle_CW.row AND jLoop = Spindle_CW.column)	THEN
			CONTINUE;
		END_IF
		
		IF buttonStatus[iLoop, jLoop] AND ((lastInput[iLoop] <> pInput[iLoop]) OR valChanged[iLoop]) THEN
			effectiveButtonStatus[iLoop, jLoop] := NOT effectiveButtonStatus[iLoop, jLoop];
			
			temp := SHL(1, jLoop);
		
			IF effectiveButtonStatus[iLoop, jLoop] THEN
				pOutput[iLoop] := pOutput[iLoop] + INT_TO_USINT(temp);
			ELSE
				pOutput[iLoop] := pOutput[iLoop] - INT_TO_USINT(temp);
			END_IF
		END_IF
		
	END_FOR
	lastInput[iLoop] := pInput[iLoop];
	valChanged[iLoop] := FALSE;
END_FOR

mSpindleButtonsHandle();

mGetButtonStatus();
END_METHOD

METHOD mParsePanelInput : BOOL
VAR_INPUT
	input   	: USINT;
	parseDigit  : INT;
END_VAR
IF ((SHR(input,parseDigit) AND 2#1) = 2#1) THEN
	mParsePanelInput := TRUE;
ELSE
	mParsePanelInput := FALSE;
END_IF
END_METHOD

METHOD mPopButton : BOOL
VAR_INPUT
	button : PanelButton;
END_VAR
IF effectiveButtonStatus[button.row, button.column] THEN
	effectiveButtonStatus[button.row, button.column]:= FALSE;
	pOutput[button.row] := pOutput[button.row] - INT_TO_USINT(SHL(1, button.column));
END_IF
END_METHOD

{attribute 'TcTypeSystem'}
{attribute 'no-analysis'}
{attribute 'c++_compatible'}
{attribute 'minimal_input_size' := '4'}
{attribute 'pack_mode' := '4'}

METHOD mPopServoButton : HRESULT
mPopButton(ServoOn);
END_METHOD

METHOD mSpecialButtonHandle : BOOL
VAR_INPUT
END_VAR
// Reset Button -- light on only when pressed and signal lasts for 5 ms
IF effectiveButtonStatus[Reset_Button.row, Reset_Button.column] THEN
	iResetCount := iResetCount + 1;
	IF iResetCount >= GlobalVar.RESET_DURATION THEN
		buttonStatus[Reset_Button.row, Reset_Button.column] := TRUE;
		pInput[Reset_Button.row] := INT_TO_USINT(SHL(1, Reset_Button.column));
		iResetCount := 0;
	END_IF
END_IF
END_METHOD

METHOD mSpindleButtonsHandle : BOOL
VAR_INPUT
END_VAR
// Spindle Stop Button -- always light on except press CW or CCW
effectiveButtonStatus[Spindle_Stop.row, Spindle_Stop.column] := NOT(effectiveButtonStatus[Spindle_CW.row, Spindle_CW.column] OR effectiveButtonStatus[Spindle_CCW.row, Spindle_CCW.column]);

IF buttonStatus[Spindle_Stop.row, Spindle_Stop.column] AND (NOT effectiveButtonStatus[Spindle_Stop.row, Spindle_Stop.column]) THEN
	effectiveButtonStatus[Spindle_Stop.row, Spindle_Stop.column] := TRUE;
	
	mPopButton(Spindle_CW);
	
	mPopButton(Spindle_CCW);
	
END_IF

IF buttonStatus[Spindle_CW.row, Spindle_CW.column] AND effectiveButtonStatus[Spindle_Stop.row, Spindle_Stop.column] AND (NOT effectiveButtonStatus[Spindle_CW.row, Spindle_CW.column]) THEN
	effectiveButtonStatus[Spindle_CW.row, Spindle_CW.column] := TRUE;
	pOutput[Spindle_CW.row] := pOutput[Spindle_CW.row] + INT_TO_USINT(SHL(1, Spindle_CW.column));
END_IF

IF buttonStatus[Spindle_CCW.row, Spindle_CCW.column] AND effectiveButtonStatus[Spindle_Stop.row, Spindle_Stop.column] AND (NOT effectiveButtonStatus[Spindle_CCW.row, Spindle_CCW.column]) THEN
	effectiveButtonStatus[Spindle_CCW.row, Spindle_CCW.column] := TRUE;
	pOutput[Spindle_CCW.row] := pOutput[Spindle_CCW.row] + INT_TO_USINT(SHL(1, Spindle_CCW.column));
END_IF

IF effectiveButtonStatus[Spindle_Stop.row, Spindle_Stop.column] AND (NOT bSpindleStopSet) THEN
	pOutput[Spindle_Stop.row] := pOutput[Spindle_Stop.row] + INT_TO_USINT(SHL(1, Spindle_Stop.column));
	bSpindleStopSet := TRUE;
END_IF

IF (NOT effectiveButtonStatus[Spindle_Stop.row, Spindle_Stop.column]) AND bSpindleStopSet THEN
	pOutput[Spindle_Stop.row] := pOutput[Spindle_Stop.row] - INT_TO_USINT(SHL(1, Spindle_Stop.column));	
	bSpindleStopSet := FALSE;
END_IF
END_METHOD

{attribute 'object_name' := 'TcQueryInterface'}
{attribute 'c++_compatible'}
{attribute 'minimal_input_size' := '4'}
{attribute 'pack_mode' := '4'}
{attribute 'show'}
{attribute 'checksuperglobal'}

METHOD TcQueryInterface : HRESULT
VAR_INPUT
	iid	: REFERENCE TO IID;
	pipItf	: POINTER TO PVOID;
END_VAR

VAR
	ipPanel : IPanelProcess;
	ipUnk : ITcUnknown;
END_VAR
IF GuidsEqual(ADR(iid), ADR(TC_GLOBAL_IID_LIST.IID_IPanelProcess)) THEN
	ipPanel := THIS^; // cast to interface pointer
	pipItf^ := ITCUNKNOWN_TO_PVOID(ipPanel);
	TcAddRef();
	TcQueryInterface := S_OK;
ELSIF GuidsEqual(ADR(iid), ADR(TC_GLOBAL_IID_LIST.IID_ITcUnknown)) THEN
	ipUnk := THIS^; // cast to interface pointer
	pipItf^ := ITCUNKNOWN_TO_PVOID(ipUnk);
	TcAddRef(); 
	TcQueryInterface := S_OK;
ELSE
	TcQueryInterface := SUPER^.TcQueryInterface(iid, pipItf);
END_IF
END_METHOD

END_FUNCTION_BLOCK

// ---- POUs/RPC_ScopeProcess.TcPOU
{attribute 'c++_compatible'}
FUNCTION_BLOCK RPC_ScopeProcess EXTENDS TcBaseModuleRegistered IMPLEMENTS IScopeProcess

// Scope Server
VAR
	fb_GenerateFileSuffixByTime : FB_GenerateFileSuffixByTime; 	// Generate file suffix by system time
	fb_ScopeServer 		  		: FB_ScopeServer; 	  			// Record .svdx file
	bScopeRun 			  		: BOOL := FALSE; 		  		// Flag of starting or stoping scope server
	fb_ExportScopeData 	  		: FB_ExportScopeData;   		// Export recorded data after finishing 
	bExportData    		  		: BOOL := FALSE; 		  		// Flag of exporting data to file
END_VAR

// Scope Data Record
fb_ScopeServer(
	bExternalTriggerEvent	:= bScopeRun , 
	sConfigFile				:= GlobalVar.RECORD_CONFIG_PATH, 
	sSaveFile				:= CONCAT(GlobalVar.SAVE_SVDX_PREFIX, fb_GenerateFileSuffixByTime.SAVE_SVDX_SUFFIX));
	
fb_ExportScopeData(
	sNetId					:= '' , 
	bExport					:= bExportData , 
	svd						:= fb_ScopeServer.sSaveFile , 
	target					:= CONCAT(GlobalVar.SAVE_CSV_PREFIX, fb_GenerateFileSuffixByTime.SAVE_CSV_SUFFIX) , 
	config					:= GlobalVar.RECORD_CONFIG_XML_PATH);

METHOD FB_reinit : BOOL
VAR_INPUT
END_VAR
SUPER^.FB_reinit();
END_METHOD

{attribute 'TcTypeSystem'}
{attribute 'no-analysis'}
{attribute 'c++_compatible'}
{attribute 'minimal_input_size' := '4'}
{attribute 'pack_mode' := '4'}
{attribute 'TcRpcEnable'}

METHOD mExportData : HRESULT
mExportData := S_FALSE;
bExportData := TRUE;
mExportData := S_OK;
END_METHOD

{attribute 'TcTypeSystem'}
{attribute 'no-analysis'}
{attribute 'c++_compatible'}
{attribute 'minimal_input_size' := '4'}
{attribute 'pack_mode' := '4'}
{attribute 'TcRpcEnable'}
METHOD mInitialize : HRESULT
mInitialize := S_FALSE;
// Get time to generate suffix of files saved by scope server
fb_GenerateFileSuffixByTime();
bExportData := FALSE;
mInitialize := S_OK;
END_METHOD

{attribute 'TcTypeSystem'}
{attribute 'no-analysis'}
{attribute 'c++_compatible'}
{attribute 'minimal_input_size' := '4'}
{attribute 'pack_mode' := '4'}
{attribute 'TcRpcEnable'}

METHOD mStartRecord : HRESULT
mStartRecord := S_FALSE;
// Start recording data
bScopeRun := TRUE;
mStartRecord := S_OK;
END_METHOD

{attribute 'TcTypeSystem'}
{attribute 'no-analysis'}
{attribute 'c++_compatible'}
{attribute 'minimal_input_size' := '4'}
{attribute 'pack_mode' := '4'}
{attribute 'TcRpcEnable'}

METHOD mStopRecord : HRESULT
mStopRecord := S_FALSE;
bScopeRun := FALSE;
mStopRecord := S_OK;
END_METHOD

{attribute 'object_name' := 'TcQueryInterface'}
{attribute 'c++_compatible'}
{attribute 'minimal_input_size' := '4'}
{attribute 'pack_mode' := '4'}
{attribute 'show'}
{attribute 'checksuperglobal'}

METHOD TcQueryInterface : HRESULT
VAR_INPUT
	iid	: REFERENCE TO IID;
	pipItf	: POINTER TO PVOID;
END_VAR

VAR
	ipScope : IScopeProcess;
	ipUnk : ITcUnknown;
END_VAR
IF GuidsEqual(ADR(iid), ADR(TC_GLOBAL_IID_LIST.IID_IScopeProcess)) THEN
	ipScope := THIS^; // cast to interface pointer
	pipItf^ := ITCUNKNOWN_TO_PVOID(ipScope);
	TcAddRef();
	TcQueryInterface := S_OK;
ELSIF GuidsEqual(ADR(iid), ADR(TC_GLOBAL_IID_LIST.IID_ITcUnknown)) THEN
	ipUnk := THIS^; // cast to interface pointer
	pipItf^ := ITCUNKNOWN_TO_PVOID(ipUnk);
	TcAddRef(); 
	TcQueryInterface := S_OK;
ELSE
	TcQueryInterface := SUPER^.TcQueryInterface(iid, pipItf);
END_IF
END_METHOD

END_FUNCTION_BLOCK
